# EPICS substitutions: nttable/supercycle/cols.substitutions
file col.template
{
    pattern {P, N}
            {$(P), 0}
            {$(P), 1}

}
